Yaskawa INFORM job: P-Y(FRONIUS).JBI

/JOB
//NAME P-Y(FRONIUS)
///FOLDERNAME INNE
//POS
///NPOS 9,9,9,0,0,0
///TOOL 0
///POSTYPE PULSE
///PULSE
C00000=10689,-51887,-13523,23832,68341,40974
C00001=27421,-99189,-31724,12111,36928,69280
C00002=-31937,-96410,-31111,21934,68258,25816
C00003=-49621,-69689,-22136,6804,86649,7543
C00004=-56079,-88978,-29119,12347,40887,68474
C00005=-52638,-51842,-13537,21996,60203,50942
C00006=-36193,-19652,6713,23256,73942,39672
C00007=-16262,-646,21476,20847,83467,29347
C00008=2736,-39680,-6551,20415,59949,54211
BC00000=103517,121620,531723
BC00001=103517,121620,531723
BC00002=103517,121620,531723
BC00003=103517,121620,531723
BC00004=103517,121620,531723
BC00005=103517,121620,531720
BC00006=103517,121620,531720
BC00007=103517,121620,531715
BC00008=103517,121620,531718
EC00000=0,0
EC00001=0,-247990
EC00002=0,-494606
EC00003=0,-742600
EC00004=0,-989436
EC00005=0,-1237020
EC00006=0,-1484034
EC00007=-1,-1731224
EC00008=0,-1978328
//INST
///DATE 2023/10/04 15:16
///ATTR SC,RW
///GROUP1 RB1,BS1
///GROUP2 ST1
NOP
MOVJ C00000 BC00000 VJ=0.78  +MOVJ EC00000 VJ=0.78
MOVJ C00001 BC00001 VJ=0.78  +MOVJ EC00001 VJ=0.78
MOVJ C00002 BC00002 VJ=0.78  +MOVJ EC00002 VJ=0.78
MOVJ C00003 BC00003 VJ=0.78  +MOVJ EC00003 VJ=0.78
MOVJ C00004 BC00004 VJ=0.78  +MOVJ EC00004 VJ=0.78
MOVJ C00005 BC00005 VJ=0.78  +MOVJ EC00005 VJ=0.78
MOVJ C00006 BC00006 VJ=0.78  +MOVJ EC00006 VJ=0.78
MOVJ C00007 BC00007 VJ=0.78  +MOVJ EC00007 VJ=0.78
MOVJ C00008 BC00008 VJ=0.78  +MOVJ EC00008 VJ=0.78
END
